# EPICS substitutions: IocAPP/Db/asic.substitutions
file db/saa.db {
    pattern {n_saa, bitrate, boardid, adschannel}
        {1, 128, 0, 1}
        {1, 128, 0, 2}
        {1, 128, 0, 3}
        {1, 128, 0, 4}
        {1, 128, 0, 5}
        {1, 128, 0, 6}
        {1, 128, 0, 7}
        {1, 128, 0, 8}
#        {1, 128, 1, 1} Iterate for number of asics
#        {1, 128, 1, 2}
#        {1, 128, 1, 3}
#        {1, 128, 1, 4}
#        {1, 128, 1, 5}
#        {1, 128, 1, 6}
#        {1, 128, 1, 7}
#        {1, 128, 1, 8}
}

file IocApp/Db/apfel.db {
   pattern {boardid, chipid, apfeldac, channel}
        {0, 1, 1,1}
        {0, 1, 2,1}
        {0, 1, 3,1}
        {0, 1, 4,1}
        {0, 2, 1,1}
        {0, 2, 2,1}
        {0, 2, 3,1}
        {0, 2, 4,1}
        {0, 3, 1,1}
        {0, 3, 2,1}
        {0, 3, 3,1}
        {0, 3, 4,1}
        {0, 4, 1,1}
        {0, 4, 2,1}
        {0, 4, 3,1}
        {0, 4, 4,1}
        {0, 1, 1,2}
        {0, 1, 2,2}
        {0, 1, 3,2}
        {0, 1, 4,2}
        {0, 2, 1,2}
        {0, 2, 2,2}
        {0, 2, 3,2}
        {0, 2, 4,2}
        {0, 3, 1,2}
        {0, 3, 2,2}
        {0, 3, 3,2}
        {0, 3, 4,2}
        {0, 4, 1,2}
        {0, 4, 2,2}
        {0, 4, 3,2}
        {0, 4, 4,2}
}
